FUNCTION_BLOCK FB_GlobalLogger EXTENDS FB_AbstractLogger
VAR 
    {attribute 'hide'}
	aEvent:						ARRAY [0..nSize - 1] OF ST_Event;
END_VAR
VAR CONSTANT 
	nSize: DINT:= 50; 
END_VAR

// https://github.com/PeterZerlauth/Tc3_Component

METHOD M_Notify
VAR_INPUT
	{attribute 'analysis' := '-33'}
	stEvent	: ST_Event;
END_VAR
VAR
	nIndex:				DINT;
	sMessage:			STRING(255);
END_VAR
IF (nIndex:=  M_Find(stEvent)) >= 0 THEN
	;
ELSE
	IF stEvent.eEventType >= SUPER^.eLogLevel THEN
		MEMCPY(ADR(aEvent[1]), ADR(aEvent[0]), DINT_TO_UDINT(SIZEOF(ST_Event) * (nSize - 1)));
		aEvent[0]:= stEvent;
		sMessage:= Concat(Concat(stEvent.sInstance, ' | fbObserver.P_Length = 0 | '), stEvent.sDefault);
		CASE stEvent.eEventType OF
			E_Event.Error:
				ADSLOGSTR( msgCtrlMask := ADSLOG_MSGTYPE_ERROR , msgFmtStr := '%s', strArg := sMessage);
			E_Event.Warning:
				ADSLOGSTR( msgCtrlMask := ADSLOG_MSGTYPE_WARN , msgFmtStr := '%s', strArg := sMessage);
			E_Event.Information:
				ADSLOGSTR( msgCtrlMask := ADSLOG_MSGTYPE_HINT , msgFmtStr := '%s', strArg := sMessage);
			E_Event.Debug:
				ADSLOGSTR( msgCtrlMask := ADSLOG_MSGTYPE_HINT, msgFmtStr := '%s', strArg := sMessage);
			E_Event.Verbose:
				ADSLOGSTR( msgCtrlMask := ADSLOG_MSGTYPE_HINT , msgFmtStr := '%s', strArg := sMessage);
		END_CASE
	END_IF
END_IF
END_METHOD

METHOD PUBLIC M_Find : DINT
VAR_INPUT
	stEvent:	ST_Event;
END_VAR
VAR 
	nIndex:		DINT;
END_VAR
// Find event in buffer
M_Find := -1;

WHILE nIndex < nSize - 1 DO
	IF (aEvent[nIndex].iSender = stEvent.iSender) AND_THEN
    	(aEvent[nIndex].eEventType = stEvent.eEventType) AND_THEN
		(aEvent[nIndex].sInstance = stEvent.sInstance) AND_THEN
		(aEvent[nIndex].sClass = stEvent.sClass) AND_THEN
		(aEvent[nIndex].sMessage = stEvent.sMessage) THEN
        M_Find := nIndex;
        RETURN;
    END_IF
	nIndex := nIndex + 1;
END_WHILE
END_METHOD

END_FUNCTION_BLOCK

(* stored: Version 1.1.0.1
   POU FB_GlobalLogger: Id {e1e358e0-2104-0577-0348-94cd81bffe81}, SpecialFunc None
   Method M_Notify: Id {92e19fe0-1284-0bd8-2857-6fa3f9525a45}
   Method M_Find: Id {f41793c9-9d9c-06d8-1e48-9d6c08695675} *)
